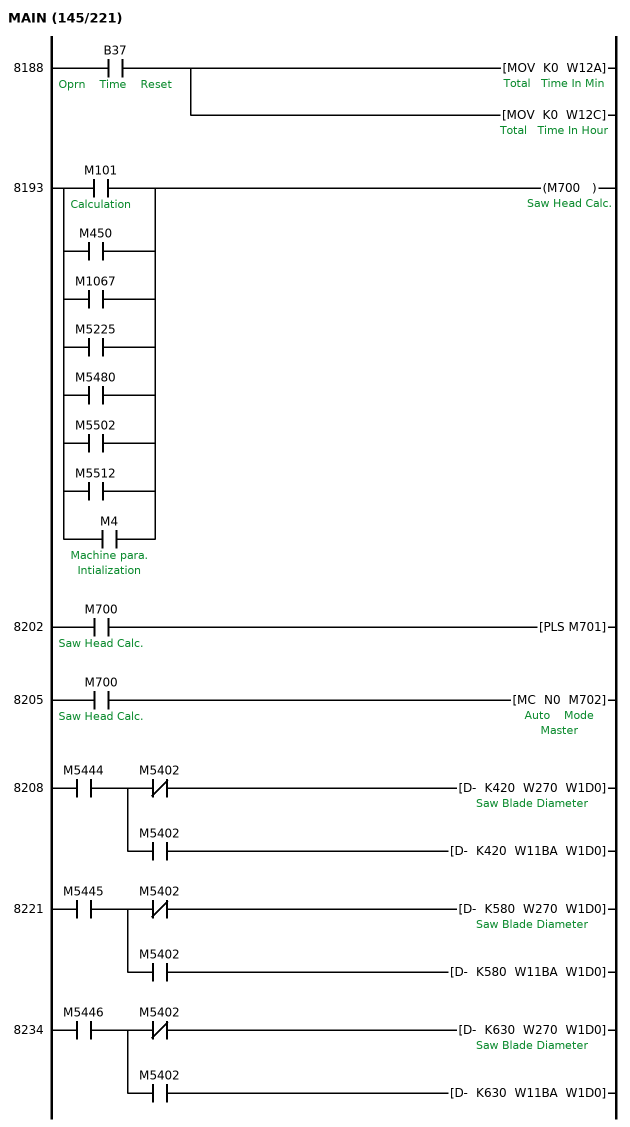
[picture p144: ladder of MAIN, rungs at steps 8188 to 8234]
8188  LD      B37  ; Oprn    Time    Reset
      MOV     K0 W12A
      MOV     K0 W12C
8193  LD      M101  ; Calculation
      OR      M450
      OR      M1067
      OR      M5225
      OR      M5480
      OR      M5502
      OR      M5512
      OR      M4  ; Machine para.   Intialization
      OUT     M700  ; Saw Head Calc.
8202  LD      M700  ; Saw Head Calc.
      PLS     M701
8205  LD      M700  ; Saw Head Calc.
      MC      N0 M702  ; Auto    Mode    Master
8208  LD      M5444
      MPS
      ANI     M5402
      D-      K420 W270 W1D0
      MPP
      AND     M5402
      D-      K420 W11BA W1D0
8221  LD      M5445
      MPS
      ANI     M5402
      D-      K580 W270 W1D0
      MPP
      AND     M5402
      D-      K580 W11BA W1D0
8234  LD      M5446
      MPS
      ANI     M5402
      D-      K630 W270 W1D0
      MPP
      AND     M5402
      D-      K630 W11BA W1D0
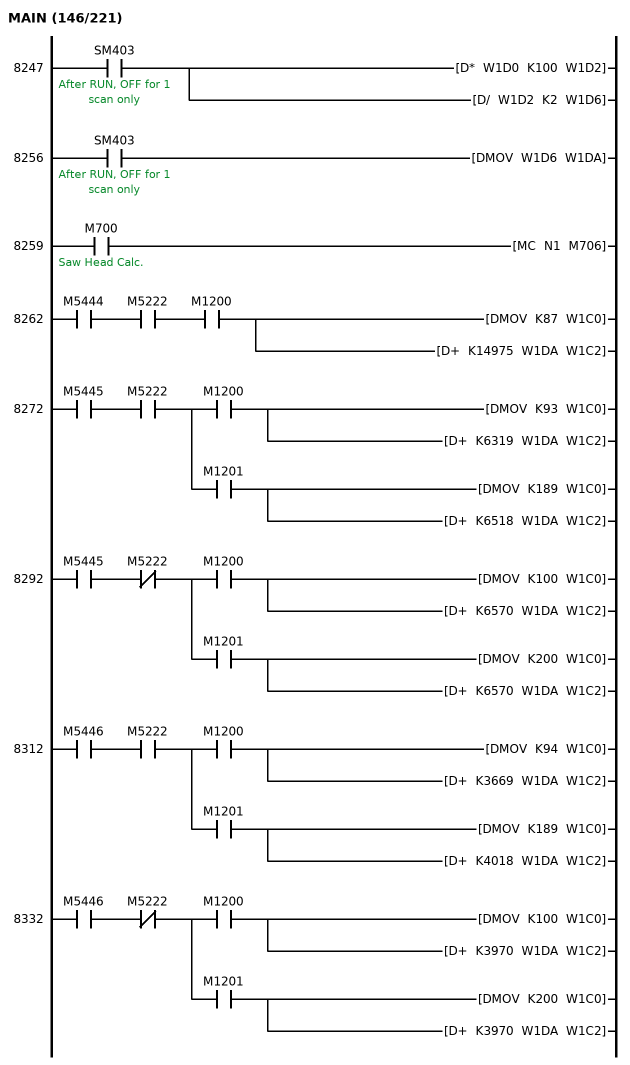
8247  LD      SM403  ; After RUN, OFF for 1 scan only
      D*      W1D0 K100 W1D2
      D/      W1D2 K2 W1D6
8256  LD      SM403  ; After RUN, OFF for 1 scan only
      DMOV    W1D6 W1DA
8259  LD      M700  ; Saw Head Calc.
      MC      N1 M706
8262  LD      M5444
      AND     M5222
      AND     M1200
      DMOV    K87 W1C0
      D+      K14975 W1DA W1C2
8272  LD      M5445
      AND     M5222
      MPS
      AND     M1200
      DMOV    K93 W1C0
      D+      K6319 W1DA W1C2
      MPP
      AND     M1201
      DMOV    K189 W1C0
      D+      K6518 W1DA W1C2
8292  LD      M5445
      ANI     M5222
      MPS
      AND     M1200
      DMOV    K100 W1C0
      D+      K6570 W1DA W1C2
      MPP
      AND     M1201
      DMOV    K200 W1C0
      D+      K6570 W1DA W1C2
8312  LD      M5446
      AND     M5222
      MPS
      AND     M1200
      DMOV    K94 W1C0
      D+      K3669 W1DA W1C2
      MPP
      AND     M1201
      DMOV    K189 W1C0
      D+      K4018 W1DA W1C2
8332  LD      M5446
      ANI     M5222
      MPS
      AND     M1200
      DMOV    K100 W1C0
      D+      K3970 W1DA W1C2
      MPP
      AND     M1201
      DMOV    K200 W1C0
      D+      K3970 W1DA W1C2
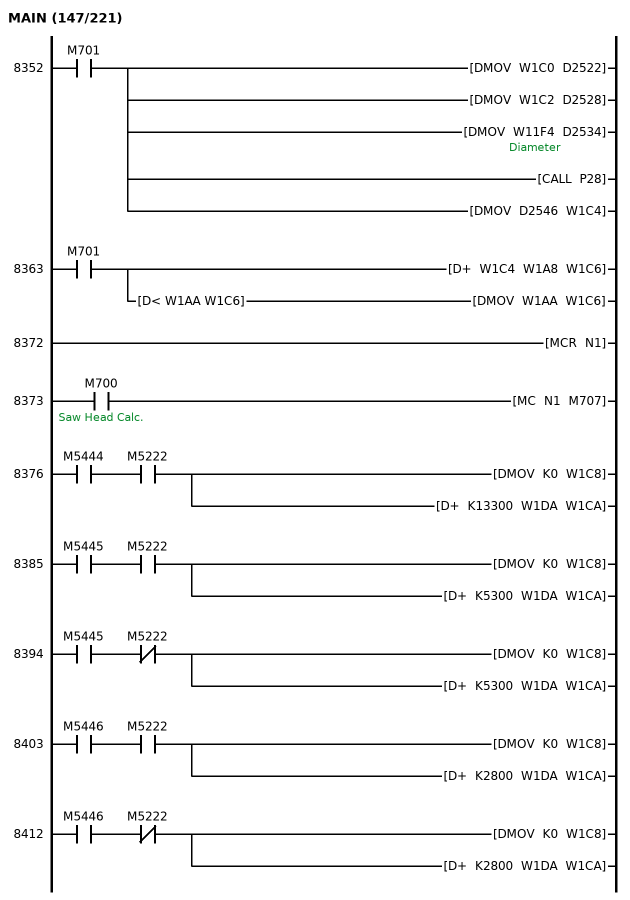
8352  LD      M701
      DMOV    W1C0 D2522
      DMOV    W1C2 D2528
      DMOV    W11F4 D2534
      CALL    P28
      DMOV    D2546 W1C4
8363  LD      M701
      D+      W1C4 W1A8 W1C6
      ANDD<   W1AA W1C6
      DMOV    W1AA W1C6
8372  MCR     N1
8373  LD      M700  ; Saw Head Calc.
      MC      N1 M707
8376  LD      M5444
      AND     M5222
      DMOV    K0 W1C8
      D+      K13300 W1DA W1CA
8385  LD      M5445
      AND     M5222
      DMOV    K0 W1C8
      D+      K5300 W1DA W1CA
8394  LD      M5445
      ANI     M5222
      DMOV    K0 W1C8
      D+      K5300 W1DA W1CA
8403  LD      M5446
      AND     M5222
      DMOV    K0 W1C8
      D+      K2800 W1DA W1CA
8412  LD      M5446
      ANI     M5222
      DMOV    K0 W1C8
      D+      K2800 W1DA W1CA
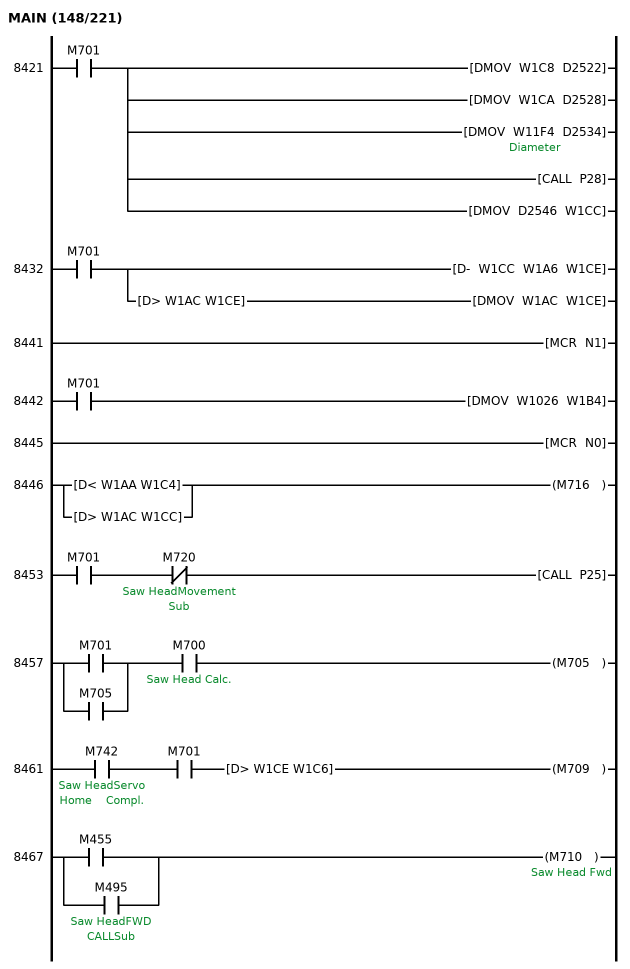
8421  LD      M701
      DMOV    W1C8 D2522
      DMOV    W1CA D2528
      DMOV    W11F4 D2534
      CALL    P28
      DMOV    D2546 W1CC
8432  LD      M701
      D-      W1CC W1A6 W1CE
      ANDD>   W1AC W1CE
      DMOV    W1AC W1CE
8441  MCR     N1
8442  LD      M701
      DMOV    W1026 W1B4
8445  MCR     N0
8446  LDD<    W1AA W1C4
      ORD>    W1AC W1CC
      OUT     M716
8453  LD      M701
      ANI     M720  ; Saw HeadMovementSub
      CALL    P25
8457  LD      M701
      OR      M705
      AND     M700  ; Saw Head Calc.
      OUT     M705
8461  LD      M742  ; Saw HeadServo   Home    Compl.
      AND     M701
      ANDD>   W1CE W1C6
      OUT     M709
8467  LD      M455
      OR      M495  ; Saw HeadFWD CALLSub
      OUT     M710  ; Saw Head Fwd
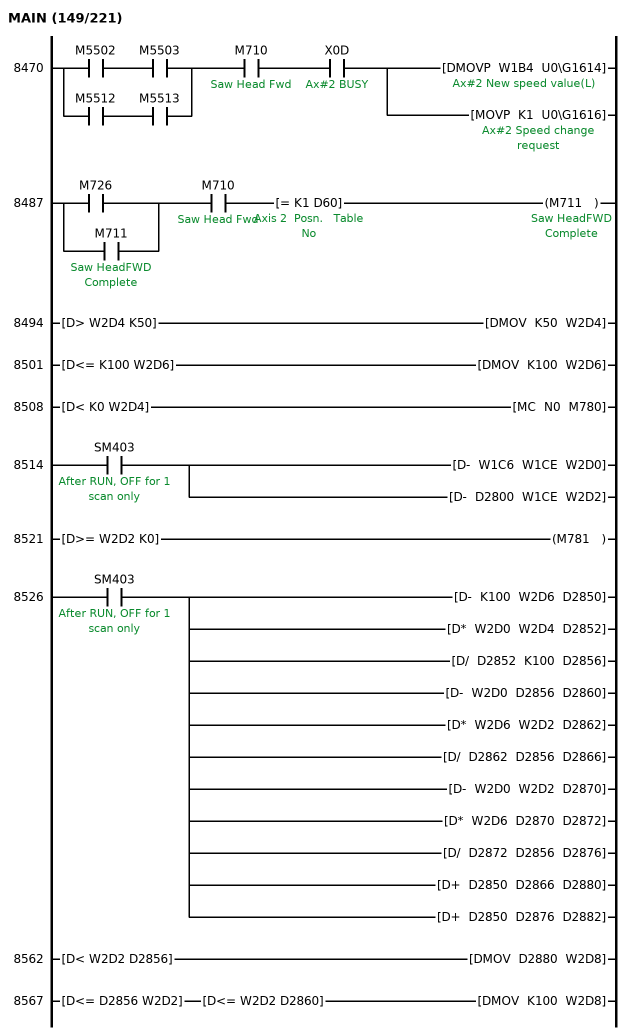
8470  LD      M5502
      AND     M5503
      LD      M5512
      AND     M5513
      ORB
      AND     M710  ; Saw Head Fwd
      AND     X0D  ; Ax#2 BUSY
      DMOVP   W1B4 U0\G1614  ; Ax#2 New speed value(L)
      MOVP    K1 U0\G1616  ; Ax#2 Speed change request
8487  LD      M726
      OR      M711  ; Saw HeadFWD     Complete
      AND     M710  ; Saw Head Fwd
      AND=    K1 D60  ; Axis 2  Posn.   Table No
      OUT     M711  ; Saw HeadFWD     Complete
8494  LDD>    W2D4 K50
      DMOV    K50 W2D4
8501  LDD<=   K100 W2D6
      DMOV    K100 W2D6
8508  LDD<    K0 W2D4
      MC      N0 M780
8514  LD      SM403  ; After RUN, OFF for 1 scan only
      D-      W1C6 W1CE W2D0
      D-      D2800 W1CE W2D2
8521  LDD>=   W2D2 K0
      OUT     M781
8526  LD      SM403  ; After RUN, OFF for 1 scan only
      D-      K100 W2D6 D2850
      D*      W2D0 W2D4 D2852
      D/      D2852 K100 D2856
      D-      W2D0 D2856 D2860
      D*      W2D6 W2D2 D2862
      D/      D2862 D2856 D2866
      D-      W2D0 W2D2 D2870
      D*      W2D6 D2870 D2872
      D/      D2872 D2856 D2876
      D+      D2850 D2866 D2880
      D+      D2850 D2876 D2882
8562  LDD<    W2D2 D2856
      DMOV    D2880 W2D8
8567  LDD<=   D2856 W2D2
      ANDD<=  W2D2 D2860
      DMOV    K100 W2D8
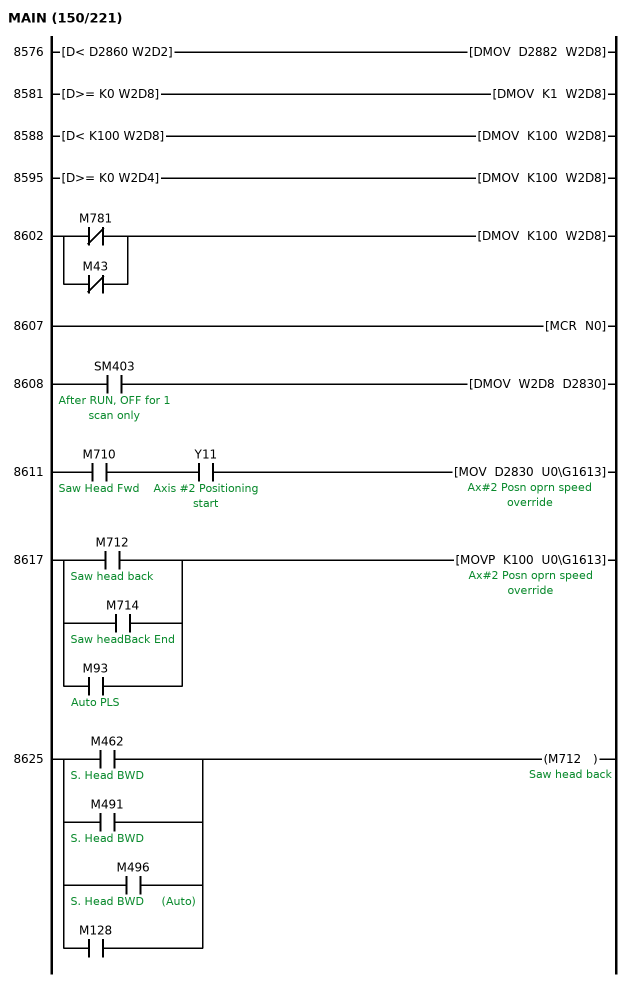
8576  LDD<    D2860 W2D2
      DMOV    D2882 W2D8
8581  LDD>=   K0 W2D8
      DMOV    K1 W2D8
8588  LDD<    K100 W2D8
      DMOV    K100 W2D8
8595  LDD>=   K0 W2D4
      DMOV    K100 W2D8
8602  LDI     M781
      ORI     M43
      DMOV    K100 W2D8
8607  MCR     N0
8608  LD      SM403  ; After RUN, OFF for 1 scan only
      DMOV    W2D8 D2830
8611  LD      M710  ; Saw Head Fwd
      AND     Y11  ; Axis #2 Positioning start
      MOV     D2830 U0\G1613  ; Ax#2 Posn oprn speed override
8617  LD      M712  ; Saw head back
      OR      M714  ; Saw headBack End
      OR      M93  ; Auto PLS
      MOVP    K100 U0\G1613
8625  LD      M462  ; S. Head BWD
      OR      M491  ; S. Head BWD
      OR      M496  ; S. Head BWD     (Auto)
      OR      M128
      OUT     M712  ; Saw head back
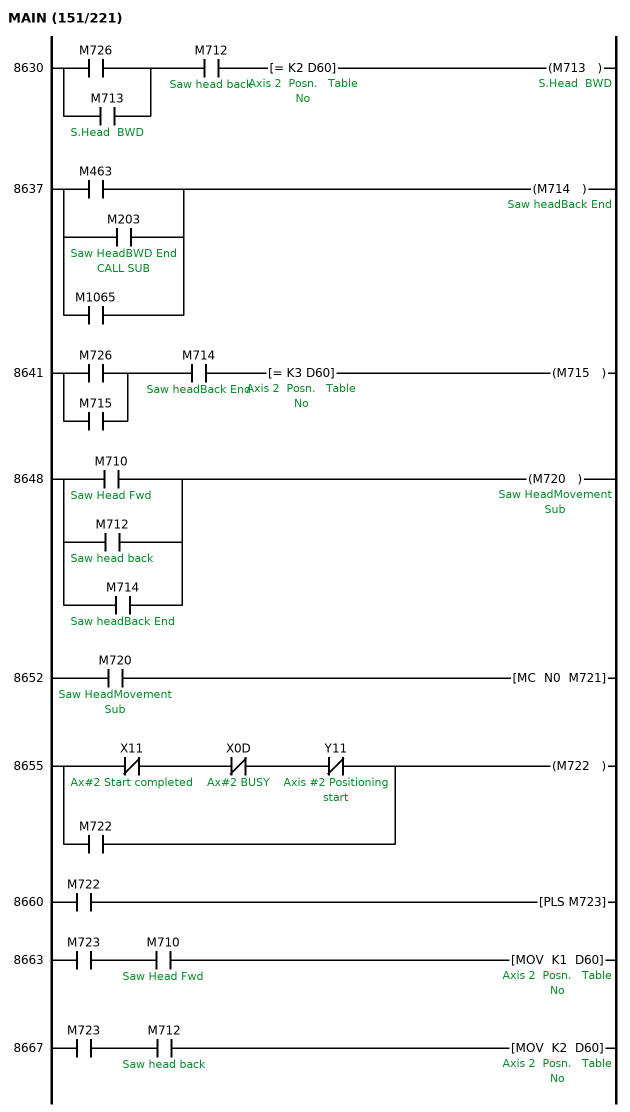
8630  LD      M726
      OR      M713  ; S.Head  BWD
      AND     M712  ; Saw head back
      AND=    K2 D60  ; Axis 2  Posn.   Table No
      OUT     M713  ; S.Head  BWD
8637  LD      M463
      OR      M203  ; Saw HeadBWD End CALL SUB
      OR      M1065
      OUT     M714  ; Saw headBack End
8641  LD      M726
      OR      M715
      AND     M714  ; Saw headBack End
      AND=    K3 D60  ; Axis 2  Posn.   Table No
      OUT     M715
8648  LD      M710  ; Saw Head Fwd
      OR      M712  ; Saw head back
      OR      M714  ; Saw headBack End
      OUT     M720  ; Saw HeadMovementSub
8652  LD      M720  ; Saw HeadMovementSub
      MC      N0 M721
8655  LDI     X11  ; Ax#2 Start completed
      ANI     X0D  ; Ax#2 BUSY
      ANI     Y11  ; Axis #2 Positioning start
      OR      M722
      OUT     M722
8660  LD      M722
      PLS     M723
8663  LD      M723
      AND     M710  ; Saw Head Fwd
      MOV     K1 D60
8667  LD      M723
      AND     M712  ; Saw head back
      MOV     K2 D60
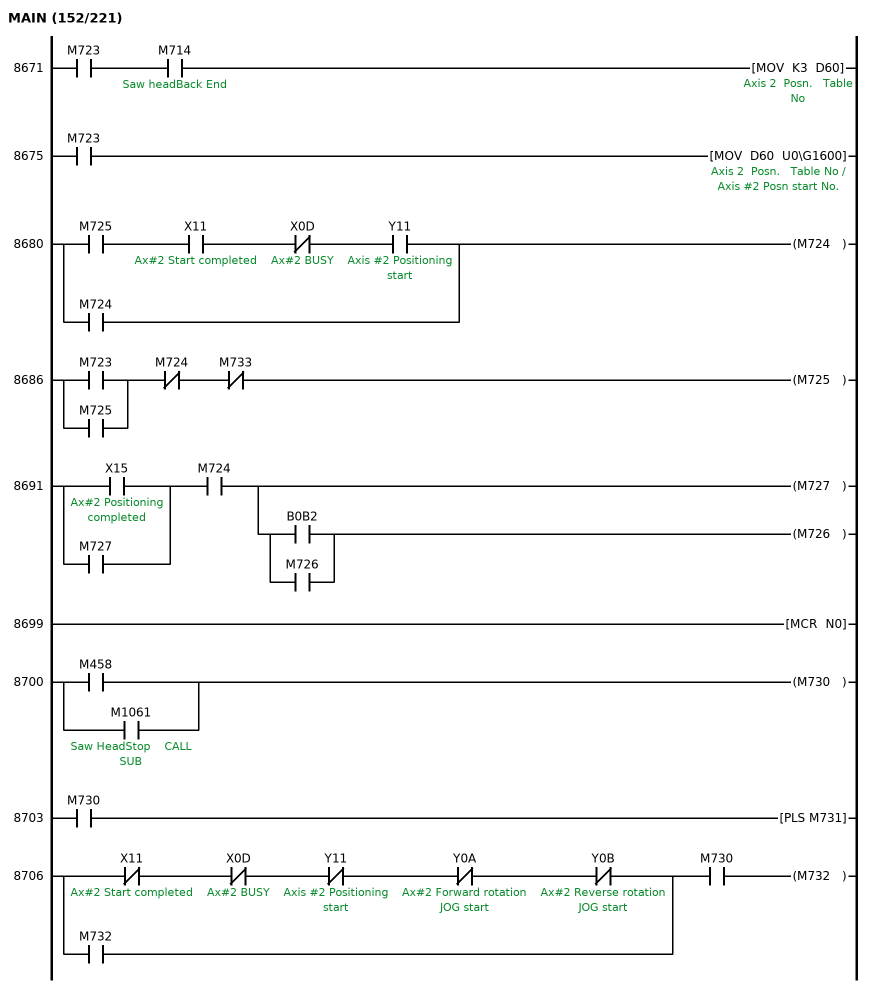
8671  LD      M723
      AND     M714  ; Saw headBack End
      MOV     K3 D60
8675  LD      M723
      MOV     D60 U0\G1600  ; Axis #2 Posn start No.
8680  LD      M725
      AND     X11  ; Ax#2 Start completed
      ANI     X0D  ; Ax#2 BUSY
      AND     Y11  ; Axis #2 Positioning start
      OR      M724
      OUT     M724
8686  LD      M723
      OR      M725
      ANI     M724
      ANI     M733
      OUT     M725
8691  LD      X15  ; Ax#2 Positioning completed
      OR      M727
      AND     M724
      OUT     M727
      LD      B0B2
      OR      M726
      ANB
      OUT     M726
8699  MCR     N0
8700  LD      M458
      OR      M1061  ; Saw HeadStop    CALL SUB
      OUT     M730
8703  LD      M730
      PLS     M731
8706  LDI     X11  ; Ax#2 Start completed
      ANI     X0D  ; Ax#2 BUSY
      ANI     Y11  ; Axis #2 Positioning start
      ANI     Y0A  ; Ax#2 Forward rotation JOG start
      ANI     Y0B  ; Ax#2 Reverse rotation JOG start
      OR      M732
      AND     M730
      OUT     M732
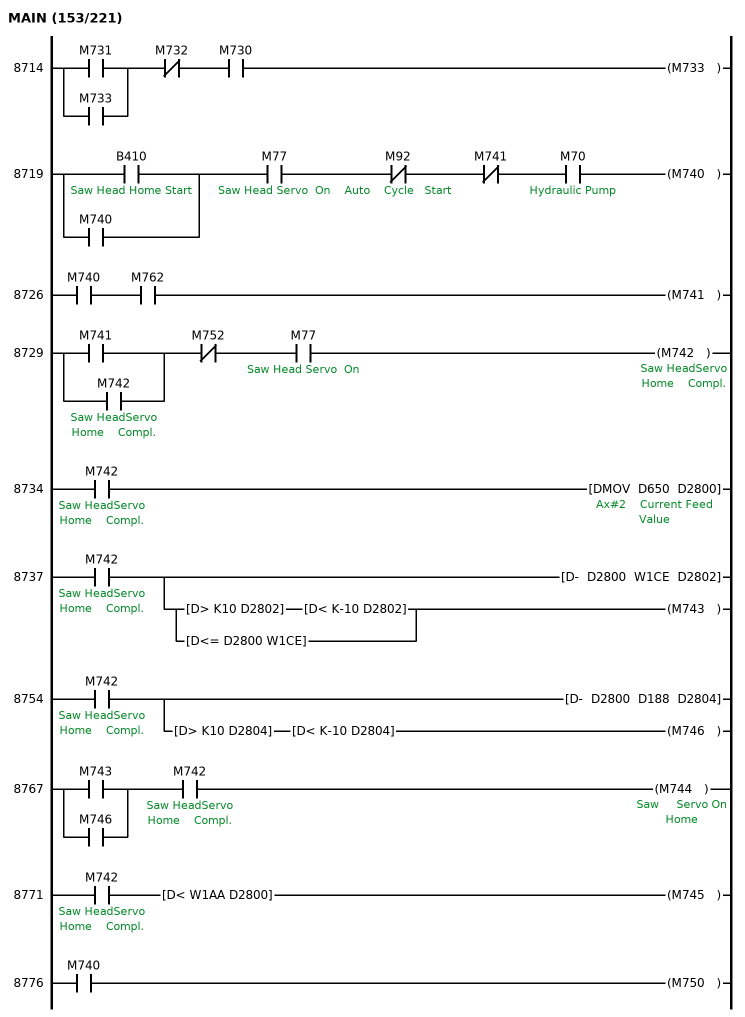
8714  LD      M731
      OR      M733
      ANI     M732
      AND     M730
      OUT     M733
8719  LD      B410  ; Saw Head Home Start
      OR      M740
      AND     M77  ; Saw Head Servo  On
      ANI     M92  ; Auto    Cycle   Start
      ANI     M741
      AND     M70  ; Hydraulic Pump
      OUT     M740
8726  LD      M740
      AND     M762
      OUT     M741
8729  LD      M741
      OR      M742  ; Saw HeadServo   Home    Compl.
      ANI     M752
      AND     M77  ; Saw Head Servo  On
      OUT     M742  ; Saw HeadServo   Home    Compl.
8734  LD      M742  ; Saw HeadServo   Home    Compl.
      DMOV    D650 D2800
8737  LD      M742  ; Saw HeadServo   Home    Compl.
      D-      D2800 W1CE D2802
      LDD>    K10 D2802
      ANDD<   K-10 D2802
      ORD<=   D2800 W1CE
      ANB
      OUT     M743
8754  LD      M742  ; Saw HeadServo   Home    Compl.
      D-      D2800 D188 D2804
      ANDD>   K10 D2804
      ANDD<   K-10 D2804
      OUT     M746
8767  LD      M743
      OR      M746
      AND     M742  ; Saw HeadServo   Home    Compl.
      OUT     M744  ; Saw     Servo On Home
8771  LD      M742  ; Saw HeadServo   Home    Compl.
      ANDD<   W1AA D2800
      OUT     M745
8776  LD      M740
      OUT     M750
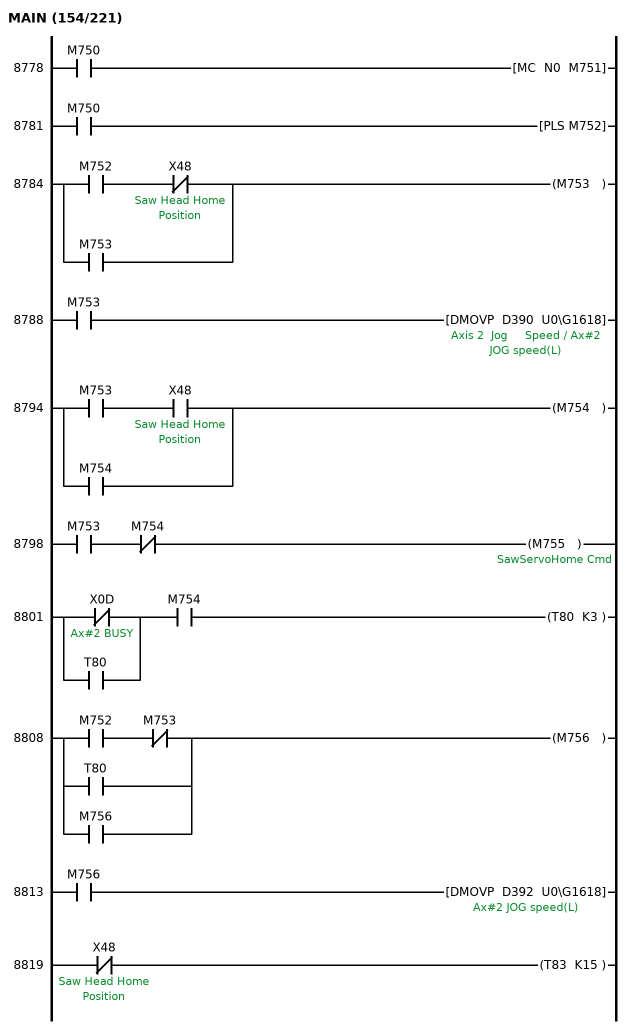
8778  LD      M750
      MC      N0 M751
8781  LD      M750
      PLS     M752
8784  LD      M752
      ANI     X48  ; Saw Head Home Position
      OR      M753
      OUT     M753
8788  LD      M753
      DMOVP   D390 U0\G1618
8794  LD      M753
      AND     X48  ; Saw Head Home Position
      OR      M754
      OUT     M754
8798  LD      M753
      ANI     M754
      OUT     M755  ; SawServoHome Cmd
8801  LDI     X0D  ; Ax#2 BUSY
      OR      T80
      AND     M754
      OUT     T80 K3
8808  LD      M752
      ANI     M753
      OR      T80
      OR      M756
      OUT     M756
8813  LD      M756
      DMOVP   D392 U0\G1618
8819  LDI     X48  ; Saw Head Home Position
      OUT     T83 K15
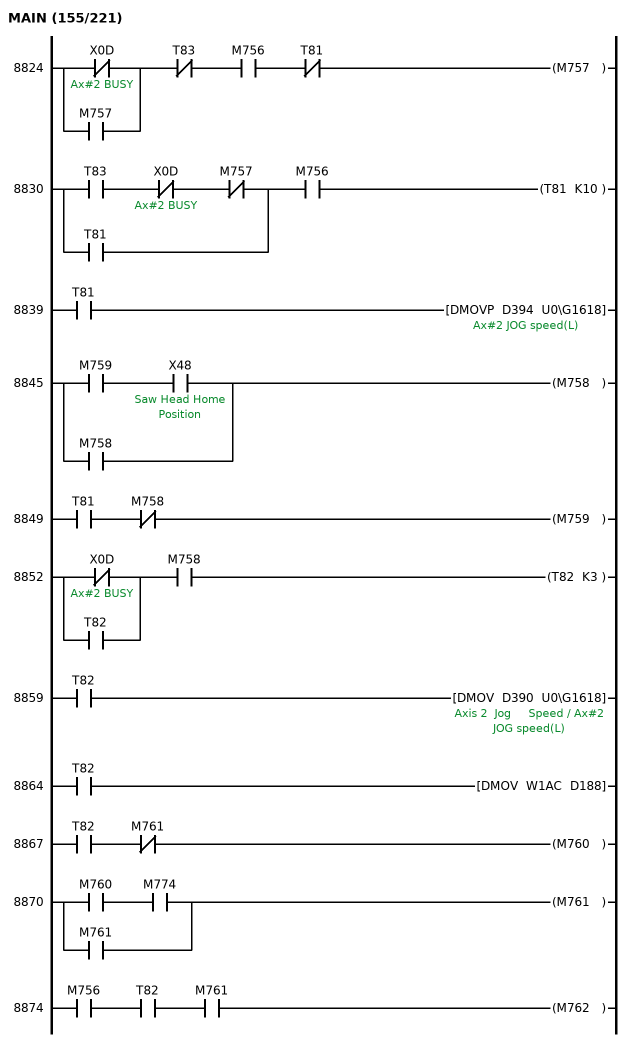
8824  LDI     X0D  ; Ax#2 BUSY
      OR      M757
      ANI     T83
      AND     M756
      ANI     T81
      OUT     M757
8830  LD      T83
      ANI     X0D  ; Ax#2 BUSY
      ANI     M757
      OR      T81
      AND     M756
      OUT     T81 K10
8839  LD      T81
      DMOVP   D394 U0\G1618
8845  LD      M759
      AND     X48  ; Saw Head Home Position
      OR      M758
      OUT     M758
8849  LD      T81
      ANI     M758
      OUT     M759
8852  LDI     X0D  ; Ax#2 BUSY
      OR      T82
      AND     M758
      OUT     T82 K3
8859  LD      T82
      DMOV    D390 U0\G1618
8864  LD      T82
      DMOV    W1AC D188
8867  LD      T82
      ANI     M761
      OUT     M760
8870  LD      M760
      AND     M774
      OR      M761
      OUT     M761
8874  LD      M756
      AND     T82
      AND     M761
      OUT     M762
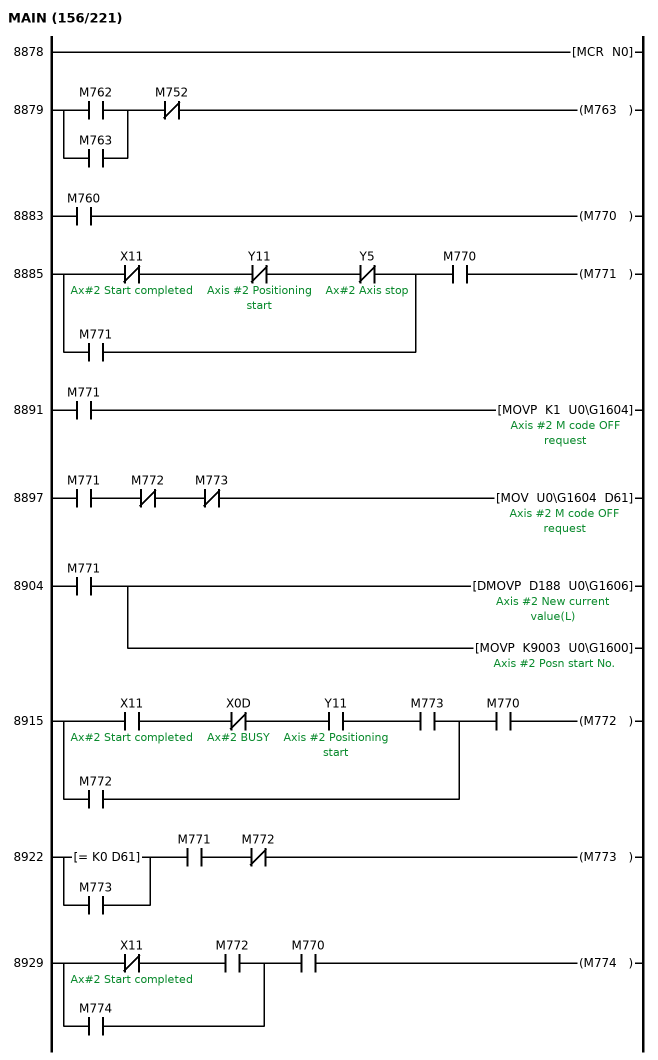
8878  MCR     N0
8879  LD      M762
      OR      M763
      ANI     M752
      OUT     M763
8883  LD      M760
      OUT     M770
8885  LDI     X11  ; Ax#2 Start completed
      ANI     Y11  ; Axis #2 Positioning start
      ANI     Y5  ; Ax#2 Axis stop
      OR      M771
      AND     M770
      OUT     M771
8891  LD      M771
      MOVP    K1 U0\G1604  ; Axis #2 M code OFF request
8897  LD      M771
      ANI     M772
      ANI     M773
      MOV     U0\G1604 D61
8904  LD      M771
      DMOVP   D188 U0\G1606  ; Axis #2 New current value(L)
      MOVP    K9003 U0\G1600
8915  LD      X11  ; Ax#2 Start completed
      ANI     X0D  ; Ax#2 BUSY
      AND     Y11  ; Axis #2 Positioning start
      AND     M773
      OR      M772
      AND     M770
      OUT     M772
8922  LD=     K0 D61
      OR      M773
      AND     M771
      ANI     M772
      OUT     M773
8929  LDI     X11  ; Ax#2 Start completed
      AND     M772
      OR      M774
      AND     M770
      OUT     M774
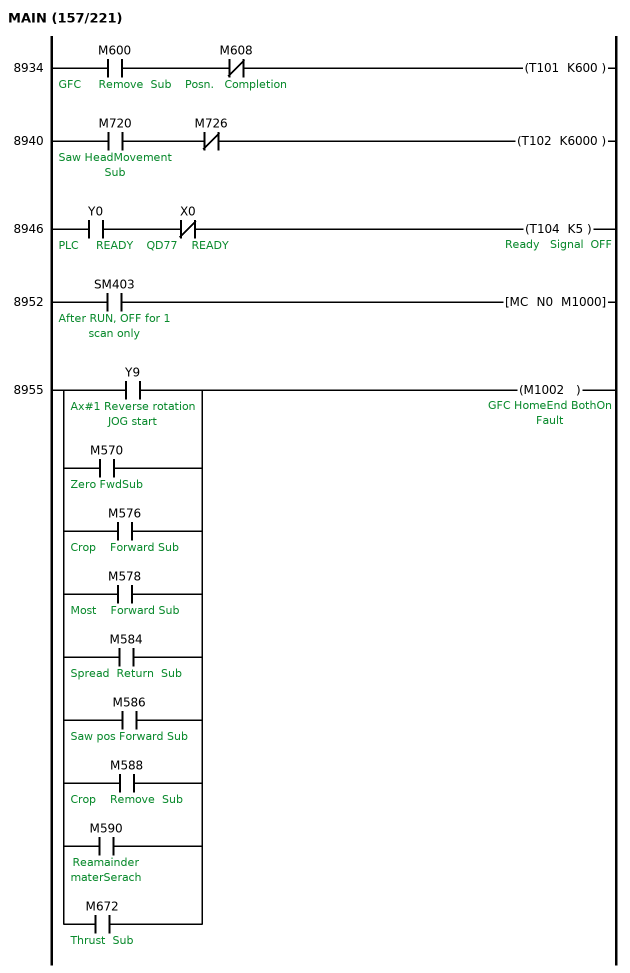
8934  LD      M600  ; GFC     Remove  Sub
      ANI     M608  ; Posn.   Completion
      OUT     T101 K600
8940  LD      M720  ; Saw HeadMovementSub
      ANI     M726
      OUT     T102 K6000
8946  LD      Y0  ; PLC     READY
      ANI     X0  ; QD77    READY
      OUT     T104 K5  ; Ready   Signal  OFF
8952  LD      SM403  ; After RUN, OFF for 1 scan only
      MC      N0 M1000
8955  LD      Y9  ; Ax#1 Reverse rotation JOG start
      OR      M570  ; Zero FwdSub
      OR      M576  ; Crop    Forward Sub
      OR      M578  ; Most    Forward Sub
      OR      M584  ; Spread  Return  Sub
      OR      M586  ; Saw pos Forward Sub
      OR      M588  ; Crop    Remove  Sub
      OR      M590  ; Reamainder materSerach
      OR      M672  ; Thrust  Sub
      OUT     M1002  ; GFC HomeEnd BothOn Fault
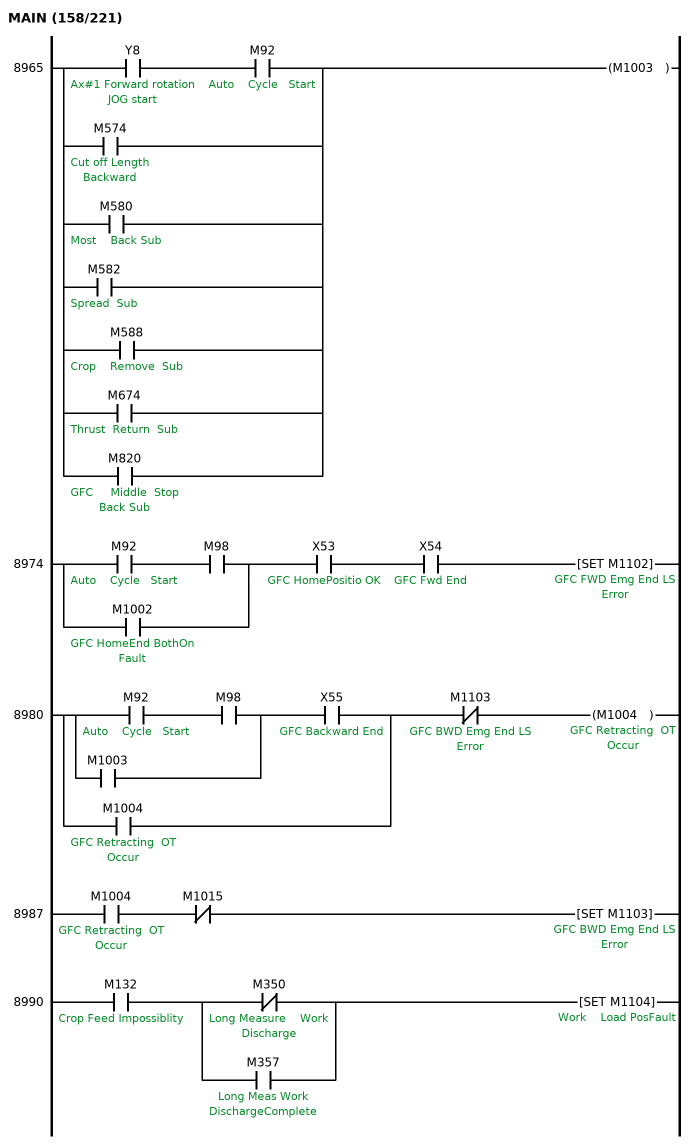
8965  LD      Y8  ; Ax#1 Forward rotation JOG start
      AND     M92  ; Auto    Cycle   Start
      OR      M574  ; Cut off Length  Backward
      OR      M580  ; Most    Back Sub
      OR      M582  ; Spread  Sub
      OR      M588  ; Crop    Remove  Sub
      OR      M674  ; Thrust  Return  Sub
      OR      M820  ; GFC     Middle  Stop    Back Sub
      OUT     M1003
8974  LD      M92  ; Auto    Cycle   Start
      AND     M98
      OR      M1002  ; GFC HomeEnd BothOn Fault
      AND     X53  ; GFC HomePositio OK
      AND     X54  ; GFC Fwd End
      SET     M1102  ; GFC FWD Emg End LS  Error
8980  LD      M92  ; Auto    Cycle   Start
      AND     M98
      OR      M1003
      AND     X55  ; GFC Backward End
      OR      M1004  ; GFC Retracting  OT Occur
      ANI     M1103  ; GFC BWD Emg End LS Error
      OUT     M1004  ; GFC Retracting  OT Occur
8987  LD      M1004  ; GFC Retracting  OT Occur
      ANI     M1015
      SET     M1103  ; GFC BWD Emg End LS Error
8990  LD      M132  ; Crop Feed Impossiblity
      LDI     M350  ; Long Measure    Work Discharge
      OR      M357  ; Long Meas Work DischargeComplete
      ANB
      SET     M1104  ; Work    Load PosFault
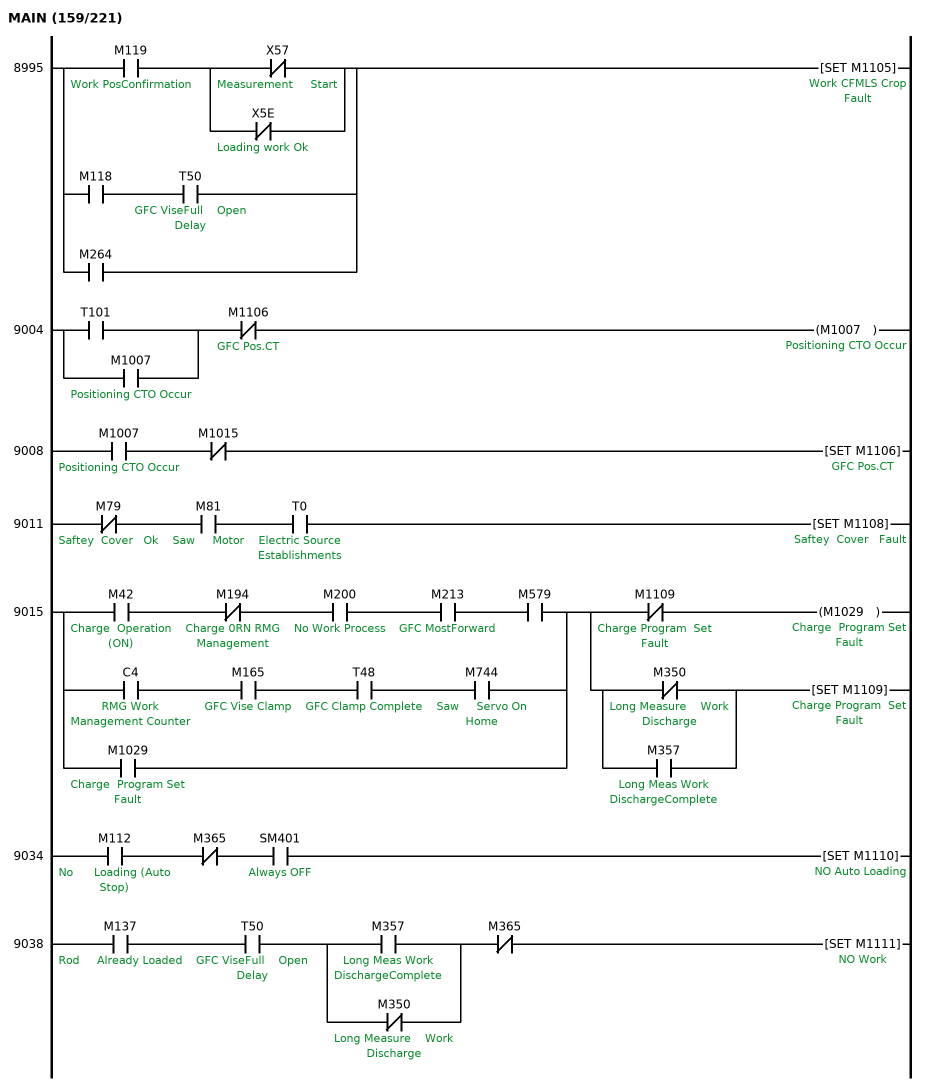
8995  LD      M119  ; Work PosConfirmation
      LDI     X57  ; Measurement     Start
      ORI     X5E  ; Loading work Ok
      ANB
      LD      M118
      AND     T50  ; GFC ViseFull    Open    Delay
      ORB
      OR      M264
      SET     M1105  ; Work CFMLS Crop Fault
9004  LD      T101
      OR      M1007  ; Positioning CTO Occur
      ANI     M1106  ; GFC Pos.CT
      OUT     M1007  ; Positioning CTO Occur
9008  LD      M1007  ; Positioning CTO Occur
      ANI     M1015
      SET     M1106  ; GFC Pos.CT
9011  LDI     M79  ; Saftey  Cover   Ok
      AND     M81  ; Saw     Motor
      AND     T0  ; Electric Source Establishments
      SET     M1108  ; Saftey  Cover   Fault
9015  LD      M42  ; Charge  Operation (ON)
      ANI     M194  ; Charge 0RN RMG  Management
      AND     M200  ; No Work Process
      AND     M213  ; GFC MostForward
      AND     M579
      LD      C4  ; RMG WorkManagement Counter
      AND     M165  ; GFC Vise Clamp
      AND     T48  ; GFC Clamp Complete
      AND     M744  ; Saw     Servo On Home
      ORB
      OR      M1029  ; Charge  Program Set     Fault
      MPS
      ANI     M1109  ; Charge Program  Set     Fault
      OUT     M1029  ; Charge  Program Set     Fault
      MPP
      LDI     M350  ; Long Measure    Work Discharge
      OR      M357  ; Long Meas Work DischargeComplete
      ANB
      SET     M1109  ; Charge Program  Set     Fault
9034  LD      M112  ; No      Loading (Auto   Stop)
      ANI     M365
      AND     SM401  ; Always OFF
      SET     M1110  ; NO Auto Loading
9038  LD      M137  ; Rod     Already Loaded
      AND     T50  ; GFC ViseFull    Open    Delay
      LD      M357  ; Long Meas Work DischargeComplete
      ORI     M350  ; Long Measure    Work Discharge
      ANB
      ANI     M365
      SET     M1111  ; NO Work
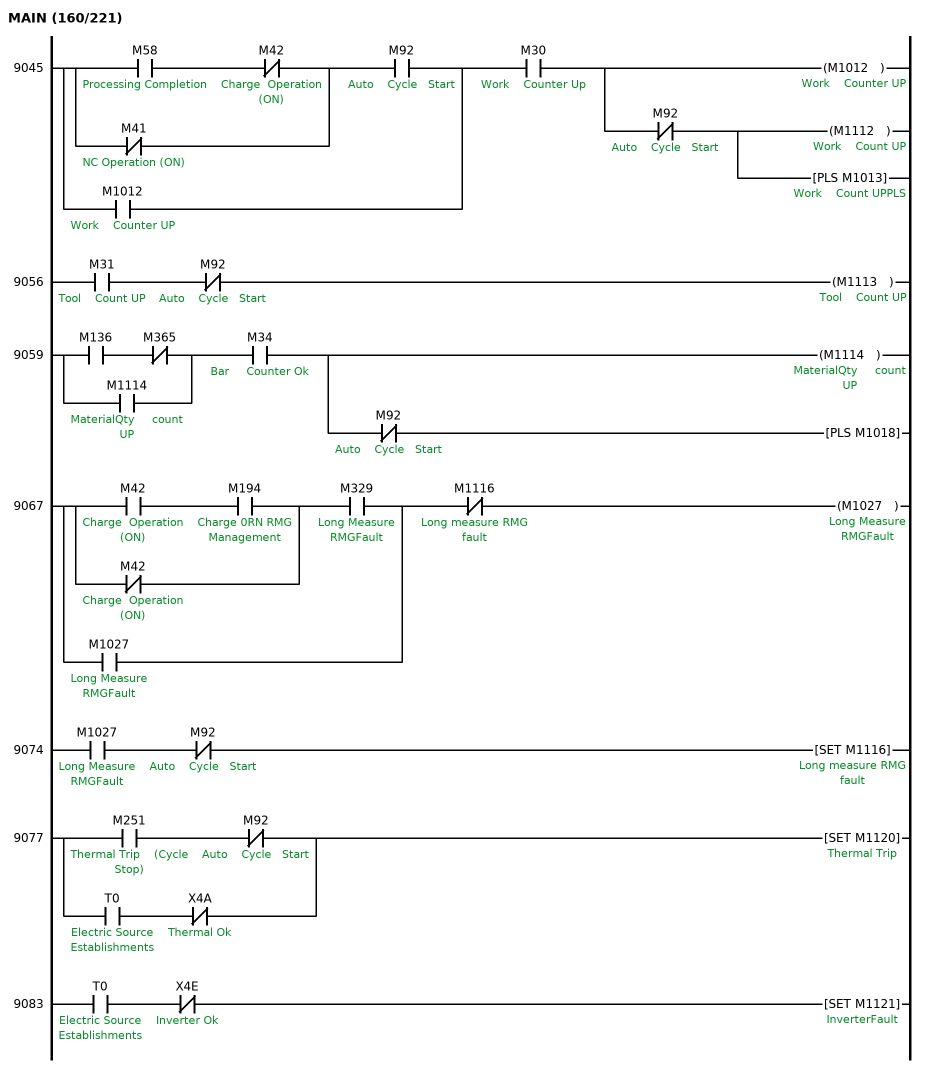
9045  LD      M58  ; Processing Completion
      ANI     M42  ; Charge  Operation (ON)
      ORI     M41  ; NC Operation (ON)
      AND     M92  ; Auto    Cycle   Start
      OR      M1012  ; Work    Counter UP
      AND     M30  ; Work    Counter Up
      OUT     M1012  ; Work    Counter UP
      ANI     M92  ; Auto    Cycle   Start
      OUT     M1112  ; Work    Count UP
      PLS     M1013  ; Work    Count UPPLS
9056  LD      M31  ; Tool    Count UP
      ANI     M92  ; Auto    Cycle   Start
      OUT     M1113  ; Tool    Count UP
9059  LD      M136
      ANI     M365
      OR      M1114  ; MaterialQty     count UP
      AND     M34  ; Bar     Counter Ok
      OUT     M1114  ; MaterialQty     count UP
      ANI     M92  ; Auto    Cycle   Start
      PLS     M1018
9067  LD      M42  ; Charge  Operation (ON)
      AND     M194  ; Charge 0RN RMG  Management
      ORI     M42  ; Charge  Operation (ON)
      AND     M329  ; Long Measure RMGFault
      OR      M1027  ; Long Measure RMGFault
      ANI     M1116  ; Long measure RMG fault
      OUT     M1027  ; Long Measure RMGFault
9074  LD      M1027  ; Long Measure RMGFault
      ANI     M92  ; Auto    Cycle   Start
      SET     M1116  ; Long measure RMG fault
9077  LD      M251  ; Thermal Trip    (Cycle  Stop)
      ANI     M92  ; Auto    Cycle   Start
      LD      T0  ; Electric Source Establishments
      ANI     X4A  ; Thermal Ok
      ORB
      SET     M1120  ; Thermal Trip
9083  LD      T0  ; Electric Source Establishments
      ANI     X4E  ; Inverter Ok
      SET     M1121  ; InverterFault
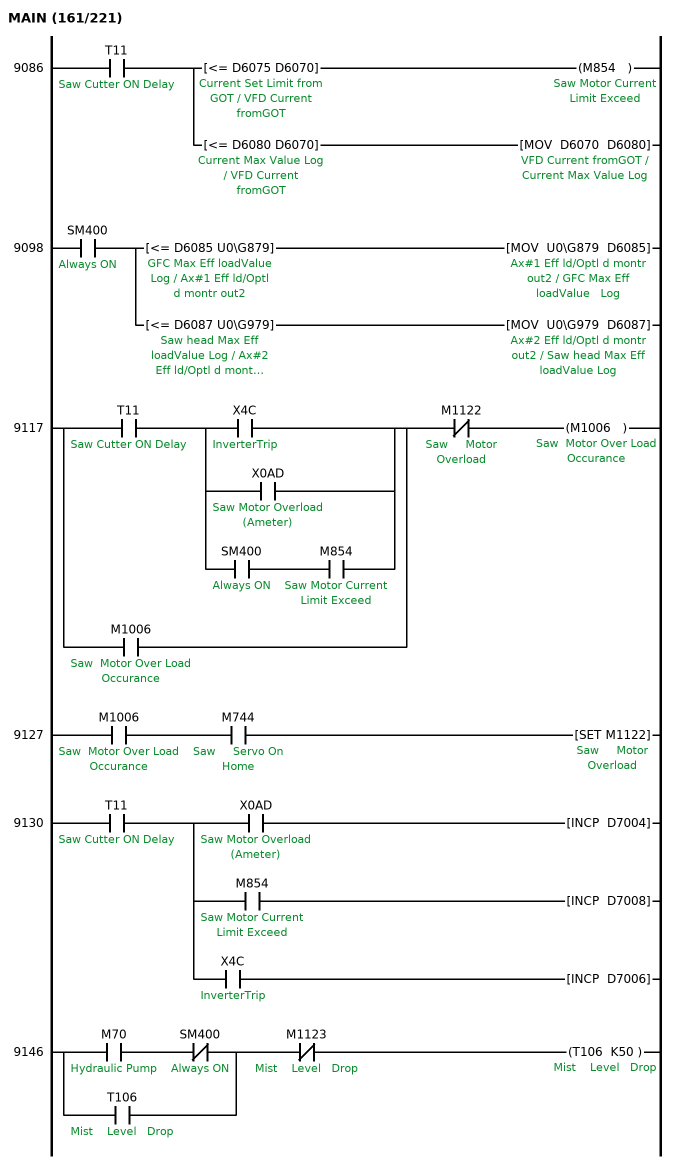
9086  LD      T11  ; Saw Cutter ON Delay
      MPS
      AND<=   D6075 D6070  ; Current Set Limit from GOT / VFD Current fromGOT
      OUT     M854  ; Saw Motor Current Limit Exceed
      MPP
      AND<=   D6080 D6070  ; Current Max Value Log / VFD Current fromGOT
      MOV     D6070 D6080
9098  LD      SM400  ; Always ON
      MPS
      AND<=   D6085 U0\G879  ; GFC Max Eff loadValue   Log / Ax#1 Eff ld/Optl d montr out2
      MOV     U0\G879 D6085
      MPP
      AND<=   D6087 U0\G979  ; Saw head Max Eff loadValue Log / Ax#2 Eff ld/Optl d montr out2
      MOV     U0\G979 D6087
9117  LD      T11  ; Saw Cutter ON Delay
      LD      X4C  ; InverterTrip
      OR      X0AD  ; Saw Motor Overload (Ameter)
      LD      SM400  ; Always ON
      AND     M854  ; Saw Motor Current Limit Exceed
      ORB
      ANB
      OR      M1006  ; Saw  Motor Over Load Occurance
      ANI     M1122  ; Saw     Motor   Overload
      OUT     M1006  ; Saw  Motor Over Load Occurance
9127  LD      M1006  ; Saw  Motor Over Load Occurance
      AND     M744  ; Saw     Servo On Home
      SET     M1122  ; Saw     Motor   Overload
9130  LD      T11  ; Saw Cutter ON Delay
      MPS
      AND     X0AD  ; Saw Motor Overload (Ameter)
      INCP    D7004
      MRD
      AND     M854  ; Saw Motor Current Limit Exceed
      INCP    D7008
      MPP
      AND     X4C  ; InverterTrip
      INCP    D7006
9146  LD      M70  ; Hydraulic Pump
      ANI     SM400  ; Always ON
      OR      T106  ; Mist    Level   Drop
      ANI     M1123  ; Mist    Level   Drop
      OUT     T106 K50  ; Mist    Level   Drop
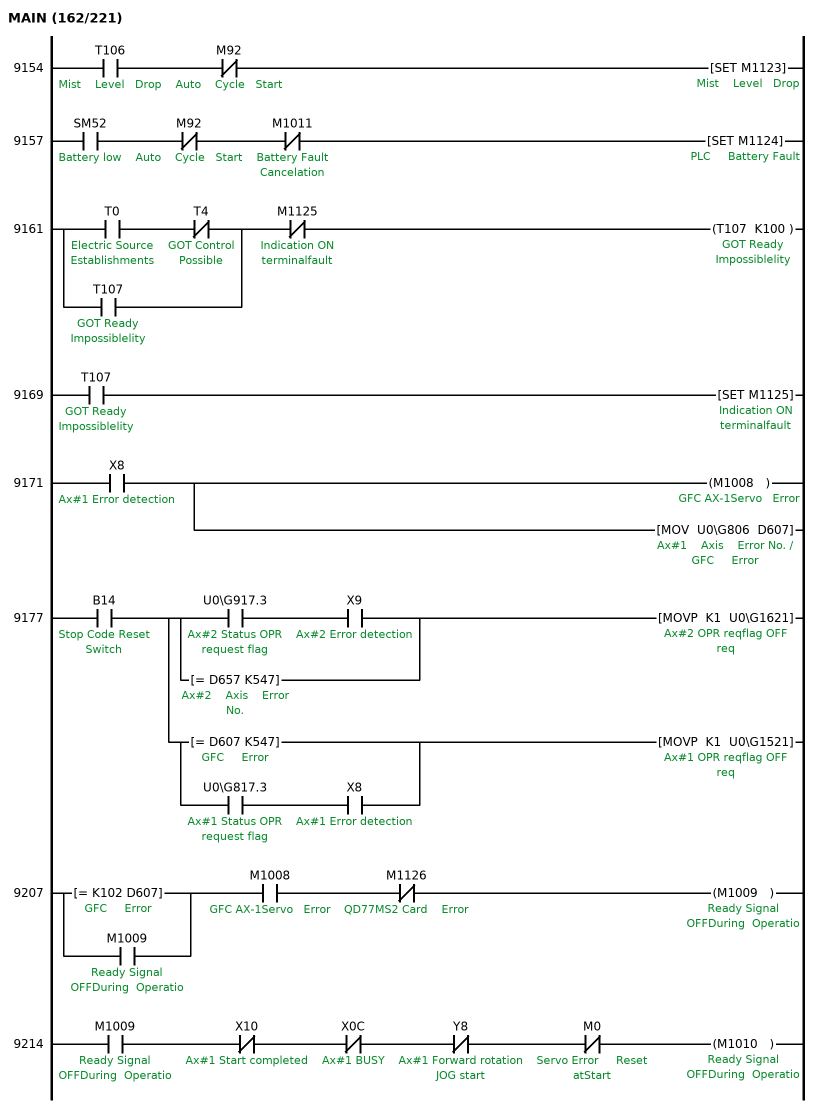
9154  LD      T106  ; Mist    Level   Drop
      ANI     M92  ; Auto    Cycle   Start
      SET     M1123  ; Mist    Level   Drop
9157  LD      SM52  ; Battery low
      ANI     M92  ; Auto    Cycle   Start
      ANI     M1011  ; Battery Fault   Cancelation
      SET     M1124  ; PLC     Battery Fault
9161  LD      T0  ; Electric Source Establishments
      ANI     T4  ; GOT Control     Possible
      OR      T107  ; GOT Ready Impossiblelity
      ANI     M1125  ; Indication ON   terminalfault
      OUT     T107 K100  ; GOT Ready Impossiblelity
9169  LD      T107  ; GOT Ready Impossiblelity
      SET     M1125  ; Indication ON   terminalfault
9171  LD      X8  ; Ax#1 Error detection
      OUT     M1008  ; GFC AX-1Servo   Error
      MOV     U0\G806 D607
9177  LD      B14  ; Stop Code Reset Switch
      MPS
      LD      U0\G917.3  ; Ax#2 Status OPR request flag
      AND     X9  ; Ax#2 Error detection
      OR=     D657 K547  ; Ax#2    Axis    Error No.
      ANB
      MOVP    K1 U0\G1621
      MPP
      LD=     D607 K547  ; GFC     Error
      LD      U0\G817.3  ; Ax#1 Status OPR request flag
      AND     X8  ; Ax#1 Error detection
      ORB
      ANB
      MOVP    K1 U0\G1521
9207  LD=     K102 D607  ; GFC     Error
      OR      M1009  ; Ready Signal OFFDuring  Operatio
      AND     M1008  ; GFC AX-1Servo   Error
      ANI     M1126  ; QD77MS2 Card    Error
      OUT     M1009  ; Ready Signal OFFDuring  Operatio
9214  LD      M1009  ; Ready Signal OFFDuring  Operatio
      ANI     X10  ; Ax#1 Start completed
      ANI     X0C  ; Ax#1 BUSY
      ANI     Y8  ; Ax#1 Forward rotation JOG start
      ANI     M0  ; Servo Error     Reset atStart
      OUT     M1010  ; Ready Signal OFFDuring  Operatio
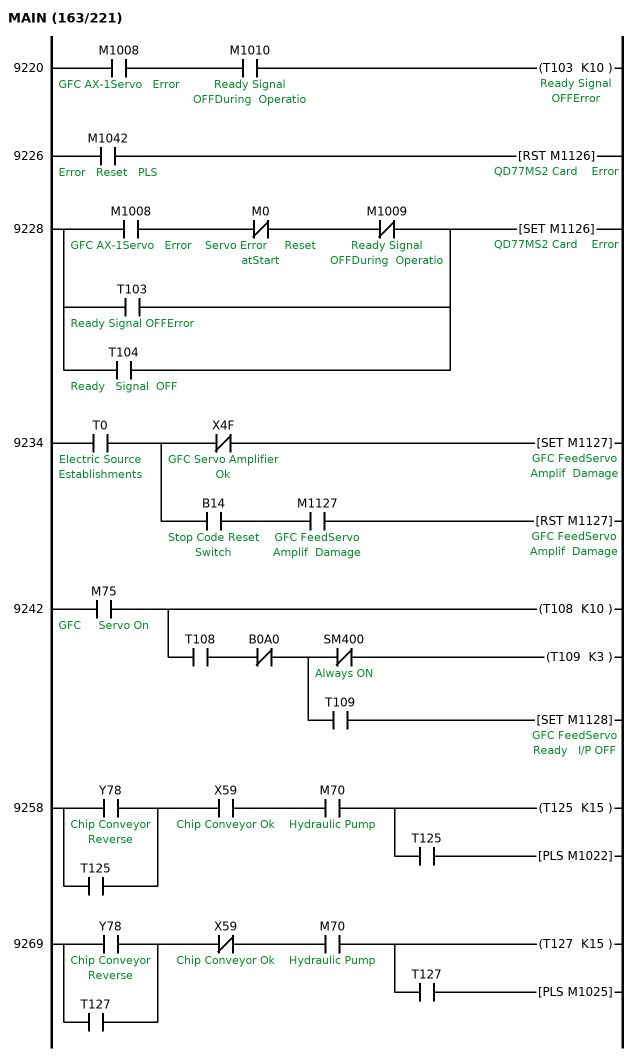
9220  LD      M1008  ; GFC AX-1Servo   Error
      AND     M1010  ; Ready Signal OFFDuring  Operatio
      OUT     T103 K10  ; Ready Signal OFFError
9226  LD      M1042  ; Error   Reset   PLS
      RST     M1126  ; QD77MS2 Card    Error
9228  LD      M1008  ; GFC AX-1Servo   Error
      ANI     M0  ; Servo Error     Reset atStart
      ANI     M1009  ; Ready Signal OFFDuring  Operatio
      OR      T103  ; Ready Signal OFFError
      OR      T104  ; Ready   Signal  OFF
      SET     M1126  ; QD77MS2 Card    Error
9234  LD      T0  ; Electric Source Establishments
      MPS
      ANI     X4F  ; GFC Servo Amplifier Ok
      SET     M1127  ; GFC FeedServo   Amplif  Damage
      MPP
      AND     B14  ; Stop Code Reset Switch
      AND     M1127  ; GFC FeedServo   Amplif  Damage
      RST     M1127  ; GFC FeedServo   Amplif  Damage
9242  LD      M75  ; GFC     Servo On
      OUT     T108 K10
      AND     T108
      ANI     B0A0
      MPS
      ANI     SM400  ; Always ON
      OUT     T109 K3
      MPP
      AND     T109
      SET     M1128  ; GFC FeedServo   Ready   I/P OFF
9258  LD      Y78  ; Chip Conveyor Reverse
      OR      T125
      AND     X59  ; Chip Conveyor Ok
      AND     M70  ; Hydraulic Pump
      OUT     T125 K15
      AND     T125
      PLS     M1022
9269  LD      Y78  ; Chip Conveyor Reverse
      OR      T127
      ANI     X59  ; Chip Conveyor Ok
      AND     M70  ; Hydraulic Pump
      OUT     T127 K15
      AND     T127
      PLS     M1025
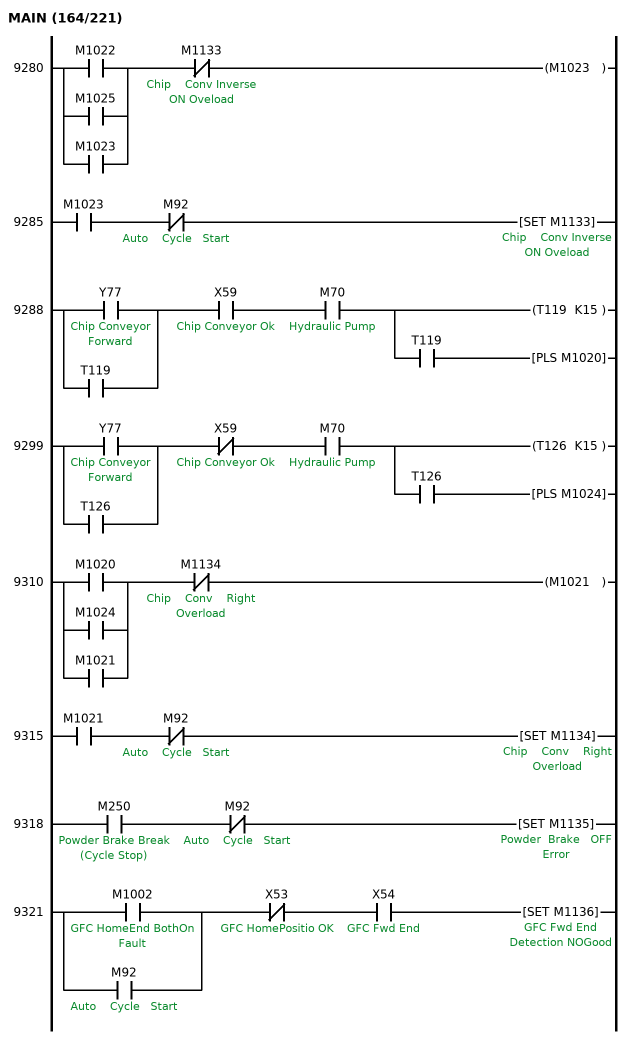
9280  LD      M1022
      OR      M1025
      OR      M1023
      ANI     M1133  ; Chip    Conv Inverse ON Oveload
      OUT     M1023
9285  LD      M1023
      ANI     M92  ; Auto    Cycle   Start
      SET     M1133  ; Chip    Conv Inverse ON Oveload
9288  LD      Y77  ; Chip Conveyor Forward
      OR      T119
      AND     X59  ; Chip Conveyor Ok
      AND     M70  ; Hydraulic Pump
      OUT     T119 K15
      AND     T119
      PLS     M1020
9299  LD      Y77  ; Chip Conveyor Forward
      OR      T126
      ANI     X59  ; Chip Conveyor Ok
      AND     M70  ; Hydraulic Pump
      OUT     T126 K15
      AND     T126
      PLS     M1024
9310  LD      M1020
      OR      M1024
      OR      M1021
      ANI     M1134  ; Chip    Conv    Right   Overload
      OUT     M1021
9315  LD      M1021
      ANI     M92  ; Auto    Cycle   Start
      SET     M1134  ; Chip    Conv    Right   Overload
9318  LD      M250  ; Powder Brake Break (Cycle Stop)
      ANI     M92  ; Auto    Cycle   Start
      SET     M1135  ; Powder  Brake   OFF     Error
9321  LD      M1002  ; GFC HomeEnd BothOn Fault
      OR      M92  ; Auto    Cycle   Start
      ANI     X53  ; GFC HomePositio OK
      AND     X54  ; GFC Fwd End
      SET     M1136  ; GFC Fwd End Detection NOGood
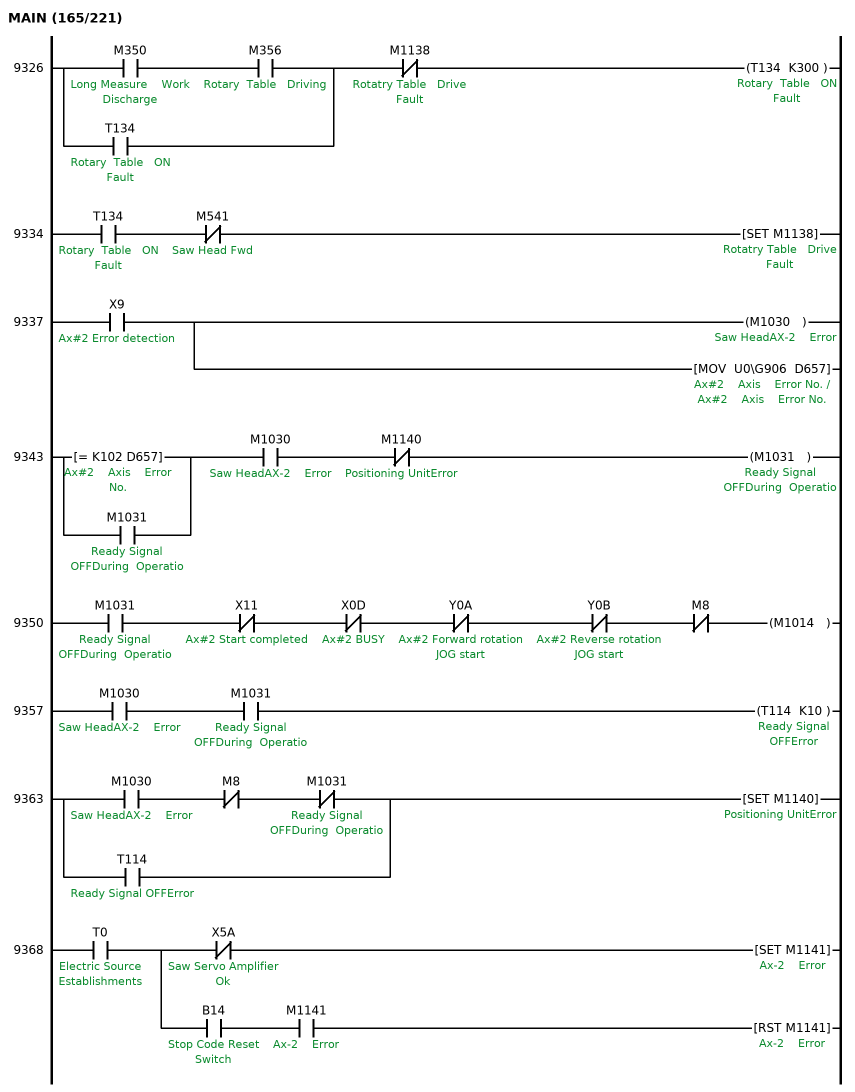
9326  LD      M350  ; Long Measure    Work Discharge
      AND     M356  ; Rotary  Table   Driving
      OR      T134  ; Rotary  Table   ON Fault
      ANI     M1138  ; Rotatry Table   Drive   Fault
      OUT     T134 K300  ; Rotary  Table   ON Fault
9334  LD      T134  ; Rotary  Table   ON Fault
      ANI     M541  ; Saw Head Fwd
      SET     M1138  ; Rotatry Table   Drive   Fault
9337  LD      X9  ; Ax#2 Error detection
      OUT     M1030  ; Saw HeadAX-2    Error
      MOV     U0\G906 D657
9343  LD=     K102 D657  ; Ax#2    Axis    Error No.
      OR      M1031  ; Ready Signal OFFDuring  Operatio
      AND     M1030  ; Saw HeadAX-2    Error
      ANI     M1140  ; Positioning UnitError
      OUT     M1031  ; Ready Signal OFFDuring  Operatio
9350  LD      M1031  ; Ready Signal OFFDuring  Operatio
      ANI     X11  ; Ax#2 Start completed
      ANI     X0D  ; Ax#2 BUSY
      ANI     Y0A  ; Ax#2 Forward rotation JOG start
      ANI     Y0B  ; Ax#2 Reverse rotation JOG start
      ANI     M8
      OUT     M1014
9357  LD      M1030  ; Saw HeadAX-2    Error
      AND     M1031  ; Ready Signal OFFDuring  Operatio
      OUT     T114 K10  ; Ready Signal OFFError
9363  LD      M1030  ; Saw HeadAX-2    Error
      ANI     M8
      ANI     M1031  ; Ready Signal OFFDuring  Operatio
      OR      T114  ; Ready Signal OFFError
      SET     M1140  ; Positioning UnitError
9368  LD      T0  ; Electric Source Establishments
      MPS
      ANI     X5A  ; Saw Servo Amplifier Ok
      SET     M1141  ; Ax-2    Error
      MPP
      AND     B14  ; Stop Code Reset Switch
      AND     M1141  ; Ax-2    Error
      RST     M1141  ; Ax-2    Error
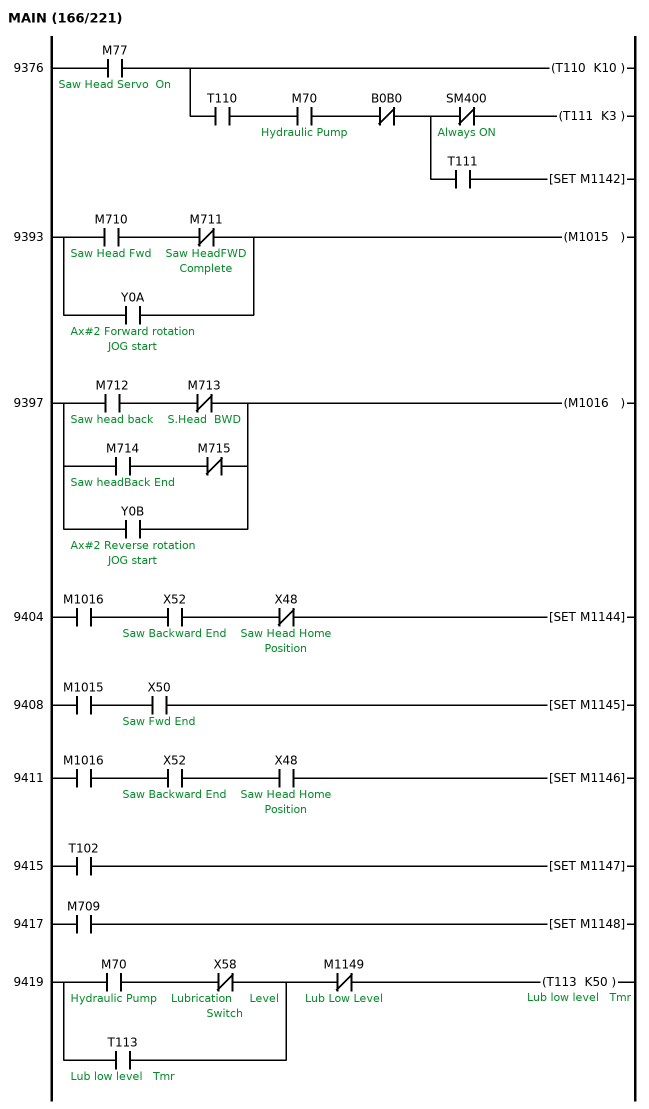
9376  LD      M77  ; Saw Head Servo  On
      OUT     T110 K10
      AND     T110
      AND     M70  ; Hydraulic Pump
      ANI     B0B0
      MPS
      ANI     SM400  ; Always ON
      OUT     T111 K3
      MPP
      AND     T111
      SET     M1142
9393  LD      M710  ; Saw Head Fwd
      ANI     M711  ; Saw HeadFWD     Complete
      OR      Y0A  ; Ax#2 Forward rotation JOG start
      OUT     M1015
9397  LD      M712  ; Saw head back
      ANI     M713  ; S.Head  BWD
      LD      M714  ; Saw headBack End
      ANI     M715
      ORB
      OR      Y0B  ; Ax#2 Reverse rotation JOG start
      OUT     M1016
9404  LD      M1016
      AND     X52  ; Saw Backward End
      ANI     X48  ; Saw Head Home Position
      SET     M1144
9408  LD      M1015
      AND     X50  ; Saw Fwd End
      SET     M1145
9411  LD      M1016
      AND     X52  ; Saw Backward End
      AND     X48  ; Saw Head Home Position
      SET     M1146
9415  LD      T102
      SET     M1147
9417  LD      M709
      SET     M1148
9419  LD      M70  ; Hydraulic Pump
      ANI     X58  ; Lubrication     Level   Switch
      OR      T113  ; Lub low level   Tmr
      ANI     M1149  ; Lub Low Level
      OUT     T113 K50  ; Lub low level   Tmr
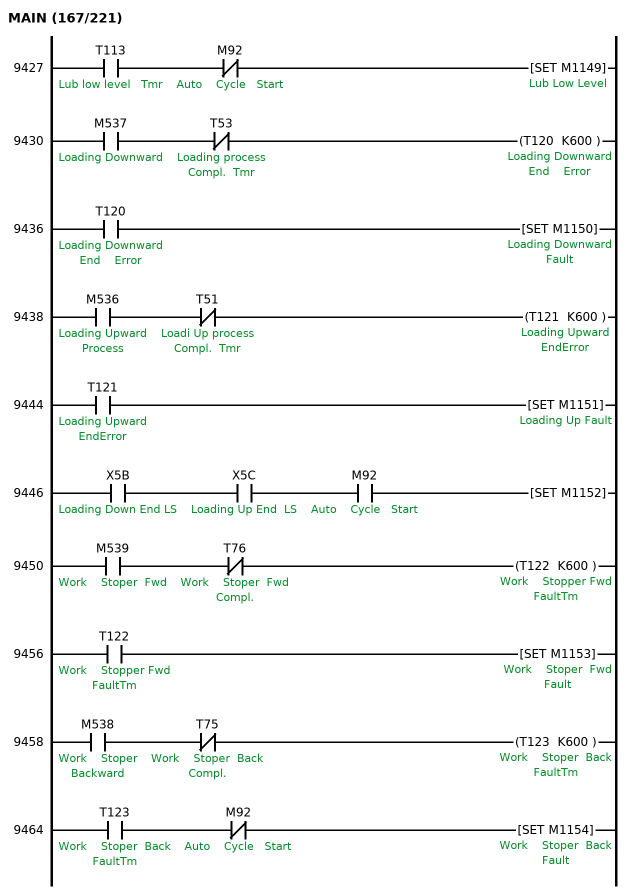
9427  LD      T113  ; Lub low level   Tmr
      ANI     M92  ; Auto    Cycle   Start
      SET     M1149  ; Lub Low Level
9430  LD      M537  ; Loading Downward
      ANI     T53  ; Loading process Compl.  Tmr
      OUT     T120 K600  ; Loading Downward End    Error
9436  LD      T120  ; Loading Downward End    Error
      SET     M1150  ; Loading Downward Fault
9438  LD      M536  ; Loading Upward  Process
      ANI     T51  ; Loadi Up process Compl.  Tmr
      OUT     T121 K600  ; Loading Upward  EndError
9444  LD      T121  ; Loading Upward  EndError
      SET     M1151  ; Loading Up Fault
9446  LD      X5B  ; Loading Down End LS
      AND     X5C  ; Loading Up End  LS
      AND     M92  ; Auto    Cycle   Start
      SET     M1152
9450  LD      M539  ; Work    Stoper  Fwd
      ANI     T76  ; Work    Stoper  Fwd     Compl.
      OUT     T122 K600  ; Work    Stopper Fwd     FaultTm
9456  LD      T122  ; Work    Stopper Fwd     FaultTm
      SET     M1153  ; Work    Stoper  Fwd     Fault
9458  LD      M538  ; Work    Stoper  Backward
      ANI     T75  ; Work    Stoper  Back    Compl.
      OUT     T123 K600  ; Work    Stoper  Back    FaultTm
9464  LD      T123  ; Work    Stoper  Back    FaultTm
      ANI     M92  ; Auto    Cycle   Start
      SET     M1154  ; Work    Stoper  Back    Fault
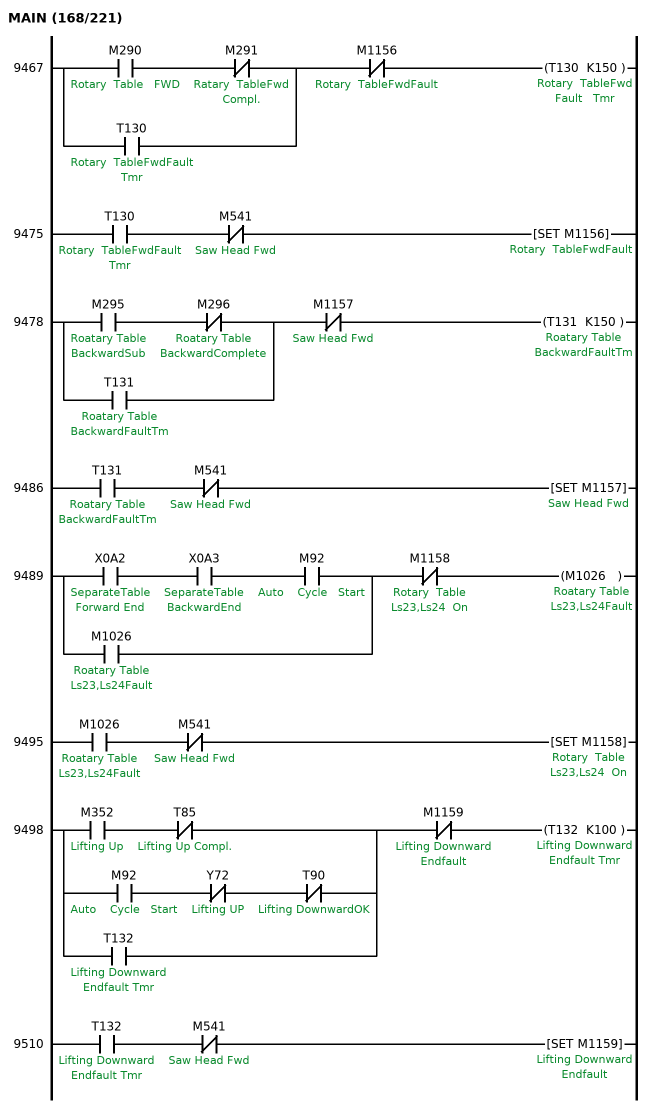
9467  LD      M290  ; Rotary  Table   FWD
      ANI     M291  ; Ratary  TableFwd Compl.
      OR      T130  ; Rotary  TableFwdFault   Tmr
      ANI     M1156  ; Rotary  TableFwdFault
      OUT     T130 K150  ; Rotary  TableFwdFault   Tmr
9475  LD      T130  ; Rotary  TableFwdFault   Tmr
      ANI     M541  ; Saw Head Fwd
      SET     M1156  ; Rotary  TableFwdFault
9478  LD      M295  ; Roatary Table   BackwardSub
      ANI     M296  ; Roatary Table   BackwardComplete
      OR      T131  ; Roatary Table   BackwardFaultTm
      ANI     M1157  ; Saw Head Fwd
      OUT     T131 K150  ; Roatary Table   BackwardFaultTm
9486  LD      T131  ; Roatary Table   BackwardFaultTm
      ANI     M541  ; Saw Head Fwd
      SET     M1157  ; Saw Head Fwd
9489  LD      X0A2  ; SeparateTable   Forward End
      AND     X0A3  ; SeparateTable   BackwardEnd
      AND     M92  ; Auto    Cycle   Start
      OR      M1026  ; Roatary Table  Ls23,Ls24Fault
      ANI     M1158  ; Rotary  Table Ls23,Ls24  On
      OUT     M1026  ; Roatary Table  Ls23,Ls24Fault
9495  LD      M1026  ; Roatary Table  Ls23,Ls24Fault
      ANI     M541  ; Saw Head Fwd
      SET     M1158  ; Rotary  Table Ls23,Ls24  On
9498  LD      M352  ; Lifting Up
      ANI     T85  ; Lifting Up Compl.
      LD      M92  ; Auto    Cycle   Start
      ANI     Y72  ; Lifting UP
      ANI     T90  ; Lifting DownwardOK
      ORB
      OR      T132  ; Lifting DownwardEndfault Tmr
      ANI     M1159  ; Lifting DownwardEndfault
      OUT     T132 K100  ; Lifting DownwardEndfault Tmr
9510  LD      T132  ; Lifting DownwardEndfault Tmr
      ANI     M541  ; Saw Head Fwd
      SET     M1159  ; Lifting DownwardEndfault
